// TIA Portal project "CERRADURA" (V11)

(* hardware
DEVICE "S7300/ET200 station_1"  SIMATIC 300-Station
   slot 0: "Perfil soporte_0"  Rail  6ES7 390-1***0-0AA0
   slot 1: "PS 307 2A_1"  PS 307 2A  6ES7 307-1BA00-0AA0
   slot 2: "PLC_1"  CPU 313C-2 DP  6ES7 313-6CF03-0AB0  V2.6
      slot 0: "Interfaz MPI_1"  MPI
      slot 1: "Interfaz DP_1"  DP
      slot 2: "DI16/DO16_1"  DI16/DO16
      slot 4: "Contaje_1"  Counter
   slot 4: "AI4/AO2 x 8bits_1"  AI4/AO2x8/8Bit  6ES7 334-0CE01-0AA0
   slot 5: "CP 343-1 Lean_1"  CP 343-1 LEAN  6GK7 343-1CX10-0XE0  V2.4
   slot 6: "CP 340 RS232C_1"  CP 340 RS232C  6ES7 340-1AH02-0AE0  V1.0
   slot 7: "CP 340 RS422/485_1"  CP 340 RS422/485  6ES7 340-1CH02-0AE0  V1.0
*)

// ===== PLC "PLC_1"  CPU 313C-2 DP =====

VAR_GLOBAL   // PLC tag table "Tabla de variables estándar"
   "1" AT %E0.0 : Bool;
   "2" AT %E0.1 : Bool;
   "3" AT %E0.2 : Bool;
   "4" AT %E0.3 : Bool;
   "5" AT %E0.4 : Bool;
   "6" AT %E0.5 : Bool;
   "7" AT %E0.6 : Bool;
   "8" AT %E0.7 : Bool;
   "9" AT %E1.0 : Bool;
   "0" AT %E1.1 : Bool;
   "#" AT %E1.2 : Bool;
   "*" AT %E1.3 : Bool;
   "Tag_1" AT %AB0 : Byte;
   "Tag_2" AT %AB1 : Byte;
   "Tag_3" AT %AB2 : Byte;
   "Tag_4" AT %AB3 : Byte;
   "Tag_5" AT %M0.0 : Bool;
   "Tag_6" AT %T0 : Timer;
   "Tag_7" AT %A0.0 : Bool;
   "Tag_8" AT %M100.1 : Bool;
   "Tag_9" AT %M100.5 : Bool;
   "Tag_10" AT %A0.1 : Bool;
   "Tag_11" AT %A0.3 : Bool;
   "Tag_12" AT %A3.1 : Bool;
END_VAR

DATA_BLOCK "AUXILIARES"   // DB1
{ S7_Optimized_Access := 'FALSE' }
VERSION : 0.1
   VAR
      FLANCOS : Array [0..70] of Bool;
      BOBINAS : Array [0..70] of Bool;
      REPRESENTACION : Array [0..3] of Byte;
      "CONTADOR H-ACTUAL" : Array [0..2] of Int;
   END_VAR
BEGIN
END_DATA_BLOCK

FUNCTION "DISPLAY UNID. MILLAR." : Void   // FC1, LAD
TITLE = DISPLAY UNIDADES DE MILLAR.
{ S7_Optimized_Access := 'FALSE' }
VERSION : 0.1
// REPRESENTARA EL NUMERO O LETRA CORRESPONDIENTE.
   VAR_OUTPUT
      "UNID. MILLAR" : Byte;
   END_VAR
   VAR_TEMP   // added for the SCL form of the ladder/FBD networks
      _w1 : Bool;
   END_VAR
BEGIN

REGION Network 1: PUESTA EN MARCHA-LETRA "C" HEX. "39"
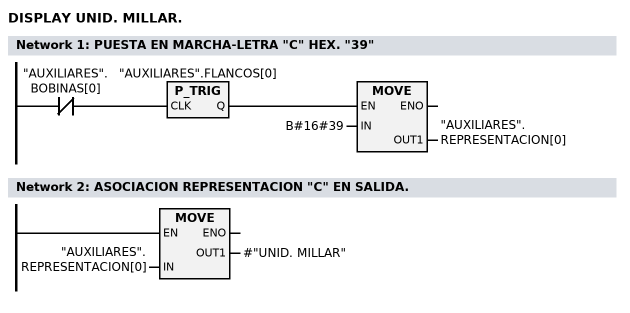
   RUNG wire#powerrail
      I_Contact( "AUXILIARES".BOBINAS[0] )
      P_Trig( "AUXILIARES".FLANCOS[0] )
      { S7_GenerateENO := "TRUE" } Move(in := B#16#39, out1 => "AUXILIARES".REPRESENTACION[0])
   END_RUNG
   // the same network as SCL:
   #_w1 := NOT "AUXILIARES".BOBINAS[0] AND NOT "AUXILIARES".FLANCOS[0];   // rising edge
   "AUXILIARES".FLANCOS[0] := NOT "AUXILIARES".BOBINAS[0];
   IF #_w1 THEN "AUXILIARES".REPRESENTACION[0] := B#16#39; END_IF;
END_REGION

REGION Network 2: ASOCIACION REPRESENTACION "C" EN SALIDA.
   RUNG wire#powerrail
      { S7_GenerateENO := "TRUE" } Move(in := "AUXILIARES".REPRESENTACION[0], out1 => #"UNID. MILLAR")
   END_RUNG
   // the same network as SCL:
   #"UNID. MILLAR" := "AUXILIARES".REPRESENTACION[0];
END_REGION

REGION Network 3: ESTARA REPRESENTADA DURANTE 30 S.
END_REGION

REGION Network 4: CAMBIO DIGITO.
END_REGION
END_FUNCTION

FUNCTION "DISPLAY CENTANAS." : Void   // FC2, LAD
TITLE = DISPLAY CENTANAS.
{ S7_Optimized_Access := 'FALSE' }
VERSION : 0.1
// REPRESENTA EL NUMERO O LETRA CORRESPONDIENTE.
   VAR_OUTPUT
      CENTANAS : Byte;
   END_VAR
   VAR_TEMP   // added for the SCL form of the ladder/FBD networks
      _w1 : Bool;
   END_VAR
BEGIN

REGION Network 1: PUESTA EN MARCHA- "0" HEX. "3F"
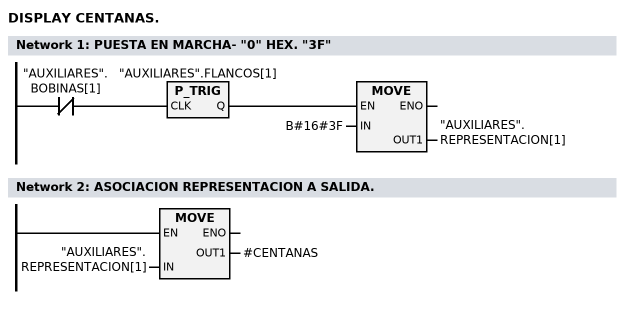
   RUNG wire#powerrail
      I_Contact( "AUXILIARES".BOBINAS[1] )
      P_Trig( "AUXILIARES".FLANCOS[1] )
      { S7_GenerateENO := "TRUE" } Move(in := B#16#3F, out1 => "AUXILIARES".REPRESENTACION[1])
   END_RUNG
   // the same network as SCL:
   #_w1 := NOT "AUXILIARES".BOBINAS[1] AND NOT "AUXILIARES".FLANCOS[1];   // rising edge
   "AUXILIARES".FLANCOS[1] := NOT "AUXILIARES".BOBINAS[1];
   IF #_w1 THEN "AUXILIARES".REPRESENTACION[1] := B#16#3F; END_IF;
END_REGION

REGION Network 2: ASOCIACION REPRESENTACION A SALIDA.
   RUNG wire#powerrail
      { S7_GenerateENO := "TRUE" } Move(in := "AUXILIARES".REPRESENTACION[1], out1 => #CENTANAS)
   END_RUNG
   // the same network as SCL:
   #CENTANAS := "AUXILIARES".REPRESENTACION[1];
END_REGION
END_FUNCTION

FUNCTION "DISPLAY DECENAS" : Void   // FC3, LAD
TITLE = DISPLAY DECENAS.
{ S7_Optimized_Access := 'FALSE' }
VERSION : 0.1
// REPRESENTA EL NUMERO O LETRA CORRESPONDIENTE.
   VAR_OUTPUT
      DECENAS : Byte;
   END_VAR
   VAR_TEMP   // added for the SCL form of the ladder/FBD networks
      _w1 : Bool;
   END_VAR
BEGIN

REGION Network 1: PUESTA EN MARCHA-"D" HEX."5E"
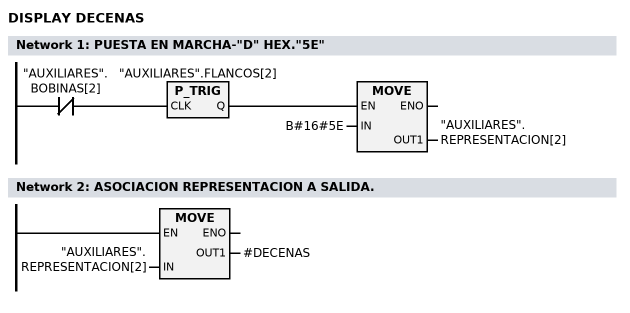
   RUNG wire#powerrail
      I_Contact( "AUXILIARES".BOBINAS[2] )
      P_Trig( "AUXILIARES".FLANCOS[2] )
      { S7_GenerateENO := "TRUE" } Move(in := B#16#5E, out1 => "AUXILIARES".REPRESENTACION[2])
   END_RUNG
   // the same network as SCL:
   #_w1 := NOT "AUXILIARES".BOBINAS[2] AND NOT "AUXILIARES".FLANCOS[2];   // rising edge
   "AUXILIARES".FLANCOS[2] := NOT "AUXILIARES".BOBINAS[2];
   IF #_w1 THEN "AUXILIARES".REPRESENTACION[2] := B#16#5E; END_IF;
END_REGION

REGION Network 2: ASOCIACION REPRESENTACION A SALIDA.
   RUNG wire#powerrail
      { S7_GenerateENO := "TRUE" } Move(in := "AUXILIARES".REPRESENTACION[2], out1 => #DECENAS)
   END_RUNG
   // the same network as SCL:
   #DECENAS := "AUXILIARES".REPRESENTACION[2];
END_REGION
END_FUNCTION

FUNCTION "DISPLAY UNIDADES." : Void   // FC4, LAD
TITLE = DISPLAY UNIDADES
{ S7_Optimized_Access := 'FALSE' }
VERSION : 0.1
// REPRESENTA EL NUMERO O LETRA CORRESPONDIENTE.
   VAR_OUTPUT
      "UNIDADES." : Byte;
   END_VAR
   VAR_TEMP   // added for the SCL form of the ladder/FBD networks
      _w1 : Bool;
   END_VAR
BEGIN

REGION Network 1: PUESTA EN MARCHA-"1" HEX. "6"
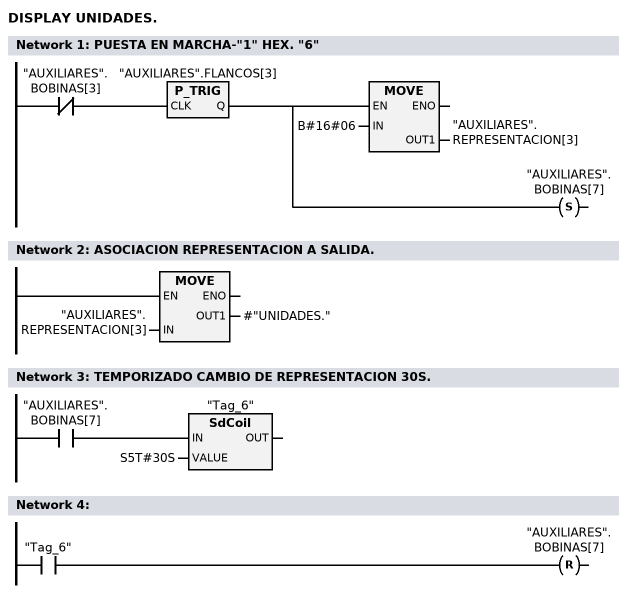
   RUNG wire#powerrail
      I_Contact( "AUXILIARES".BOBINAS[3] )
      P_Trig( "AUXILIARES".FLANCOS[3] )
      wire#w1
      { S7_GenerateENO := "TRUE" } Move(in := B#16#06, out1 => "AUXILIARES".REPRESENTACION[3])
   END_RUNG
   RUNG wire#w1
      S_Coil( "AUXILIARES".BOBINAS[7] )
   END_RUNG
   // the same network as SCL:
   #_w1 := NOT "AUXILIARES".BOBINAS[3] AND NOT "AUXILIARES".FLANCOS[3];   // rising edge
   "AUXILIARES".FLANCOS[3] := NOT "AUXILIARES".BOBINAS[3];
   IF #_w1 THEN
       "AUXILIARES".REPRESENTACION[3] := B#16#06;
       "AUXILIARES".BOBINAS[7] := TRUE;
   END_IF;
END_REGION

REGION Network 2: ASOCIACION REPRESENTACION A SALIDA.
   RUNG wire#powerrail
      { S7_GenerateENO := "TRUE" } Move(in := "AUXILIARES".REPRESENTACION[3], out1 => #"UNIDADES.")
   END_RUNG
   // the same network as SCL:
   #"UNIDADES." := "AUXILIARES".REPRESENTACION[3];
END_REGION

REGION Network 3: TEMPORIZADO CAMBIO DE REPRESENTACION 30S.
   // no SCL statement known for SdCoil: written as a call
   SdCoil(in := "AUXILIARES".BOBINAS[7], value := S5T#30S, operand := "Tag_6");
END_REGION

REGION Network 4
   RUNG wire#powerrail
      Contact( "Tag_6" )
      R_Coil( "AUXILIARES".BOBINAS[7] )
   END_RUNG
   // the same network as SCL:
   IF "Tag_6" THEN "AUXILIARES".BOBINAS[7] := FALSE; END_IF;
END_REGION
END_FUNCTION

FUNCTION "HORA ACTUAL" : Void   // FC5, LAD
TITLE = HORA ACTUAL.
{ S7_Optimized_Access := 'FALSE' }
VERSION : 0.1
// APARECE EN LOS DISPLAY POR ORDEN DE IZQUIERDA A DERECHA EN FORMATO 24 HORAS.SE REPRESENTA DESPUES DE "COD1" Y PERMANECE 60S
   VAR_TEMP   // added for the SCL form of the ladder/FBD networks
      _w1 : Bool;
      _w2 : Bool;
   END_VAR
BEGIN

REGION Network 1: CONTADOR DE SEGUNDOS.
   // MARCA DE CICLO M100.5 1S A 0N -1S A OFF.
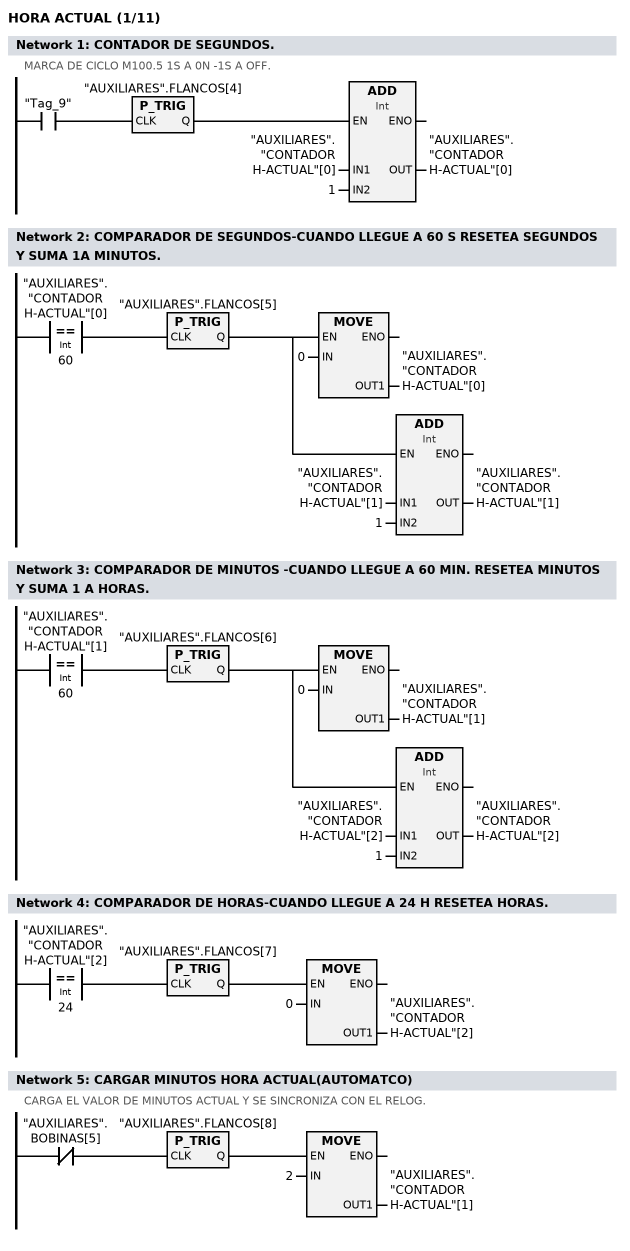
   RUNG wire#powerrail
      Contact( "Tag_9" )
      P_Trig( "AUXILIARES".FLANCOS[4] )
      { S7_Templates := "SrcType := Int"; S7_GenerateENO := "TRUE" } Add(in1 := "AUXILIARES"."CONTADOR H-ACTUAL"[0], in2 := 1, out => "AUXILIARES"."CONTADOR H-ACTUAL"[0])
   END_RUNG
   // the same network as SCL:
   #_w1 := "Tag_9" AND NOT "AUXILIARES".FLANCOS[4];   // rising edge
   "AUXILIARES".FLANCOS[4] := "Tag_9";
   IF #_w1 THEN "AUXILIARES"."CONTADOR H-ACTUAL"[0] := "AUXILIARES"."CONTADOR H-ACTUAL"[0] + 1; END_IF;
END_REGION

REGION Network 2: COMPARADOR DE SEGUNDOS-CUANDO LLEGUE A 60 S RESETEA SEGUNDOS Y SUMA 1A MINUTOS.
   RUNG wire#powerrail
      { S7_Templates := "SrcType := Int" } EQ_Contact(in1 := "AUXILIARES"."CONTADOR H-ACTUAL"[0], in2 := 60)
      P_Trig( "AUXILIARES".FLANCOS[5] )
      wire#w1
      { S7_GenerateENO := "TRUE" } Move(in := 0, out1 => "AUXILIARES"."CONTADOR H-ACTUAL"[0])
   END_RUNG
   RUNG wire#w1
      { S7_Templates := "SrcType := Int"; S7_GenerateENO := "TRUE" } Add(in1 := "AUXILIARES"."CONTADOR H-ACTUAL"[1], in2 := 1, out => "AUXILIARES"."CONTADOR H-ACTUAL"[1])
   END_RUNG
   // the same network as SCL:
   #_w1 := "AUXILIARES"."CONTADOR H-ACTUAL"[0] = 60;
   #_w2 := #_w1 AND NOT "AUXILIARES".FLANCOS[5];   // rising edge
   "AUXILIARES".FLANCOS[5] := #_w1;
   IF #_w2 THEN
       "AUXILIARES"."CONTADOR H-ACTUAL"[0] := 0;
       "AUXILIARES"."CONTADOR H-ACTUAL"[1] := "AUXILIARES"."CONTADOR H-ACTUAL"[1] + 1;
   END_IF;
END_REGION

REGION Network 3: COMPARADOR DE MINUTOS -CUANDO LLEGUE A 60 MIN. RESETEA MINUTOS Y SUMA 1 A HORAS.
   RUNG wire#powerrail
      { S7_Templates := "SrcType := Int" } EQ_Contact(in1 := "AUXILIARES"."CONTADOR H-ACTUAL"[1], in2 := 60)
      P_Trig( "AUXILIARES".FLANCOS[6] )
      wire#w1
      { S7_GenerateENO := "TRUE" } Move(in := 0, out1 => "AUXILIARES"."CONTADOR H-ACTUAL"[1])
   END_RUNG
   RUNG wire#w1
      { S7_Templates := "SrcType := Int"; S7_GenerateENO := "TRUE" } Add(in1 := "AUXILIARES"."CONTADOR H-ACTUAL"[2], in2 := 1, out => "AUXILIARES"."CONTADOR H-ACTUAL"[2])
   END_RUNG
   // the same network as SCL:
   #_w1 := "AUXILIARES"."CONTADOR H-ACTUAL"[1] = 60;
   #_w2 := #_w1 AND NOT "AUXILIARES".FLANCOS[6];   // rising edge
   "AUXILIARES".FLANCOS[6] := #_w1;
   IF #_w2 THEN
       "AUXILIARES"."CONTADOR H-ACTUAL"[1] := 0;
       "AUXILIARES"."CONTADOR H-ACTUAL"[2] := "AUXILIARES"."CONTADOR H-ACTUAL"[2] + 1;
   END_IF;
END_REGION

REGION Network 4: COMPARADOR DE HORAS-CUANDO LLEGUE A 24 H RESETEA HORAS.
   RUNG wire#powerrail
      { S7_Templates := "SrcType := Int" } EQ_Contact(in1 := "AUXILIARES"."CONTADOR H-ACTUAL"[2], in2 := 24)
      P_Trig( "AUXILIARES".FLANCOS[7] )
      { S7_GenerateENO := "TRUE" } Move(in := 0, out1 => "AUXILIARES"."CONTADOR H-ACTUAL"[2])
   END_RUNG
   // the same network as SCL:
   #_w1 := "AUXILIARES"."CONTADOR H-ACTUAL"[2] = 24;
   #_w2 := #_w1 AND NOT "AUXILIARES".FLANCOS[7];   // rising edge
   "AUXILIARES".FLANCOS[7] := #_w1;
   IF #_w2 THEN "AUXILIARES"."CONTADOR H-ACTUAL"[2] := 0; END_IF;
END_REGION

REGION Network 5: CARGAR MINUTOS HORA ACTUAL(AUTOMATCO)
   // CARGA EL VALOR DE MINUTOS ACTUAL Y SE SINCRONIZA CON EL RELOG.
   RUNG wire#powerrail
      I_Contact( "AUXILIARES".BOBINAS[5] )
      P_Trig( "AUXILIARES".FLANCOS[8] )
      { S7_GenerateENO := "TRUE" } Move(in := 2, out1 => "AUXILIARES"."CONTADOR H-ACTUAL"[1])
   END_RUNG
   // the same network as SCL:
   #_w1 := NOT "AUXILIARES".BOBINAS[5] AND NOT "AUXILIARES".FLANCOS[8];   // rising edge
   "AUXILIARES".FLANCOS[8] := NOT "AUXILIARES".BOBINAS[5];
   IF #_w1 THEN "AUXILIARES"."CONTADOR H-ACTUAL"[1] := 2; END_IF;
END_REGION

REGION Network 6: CARGAR HORAS HORA ACTUAL(AUTOMATICO).
   // CARGA EL VALOR DE HORAS ACTUAL Y SE SINCRONIZA CON EL RELOG.
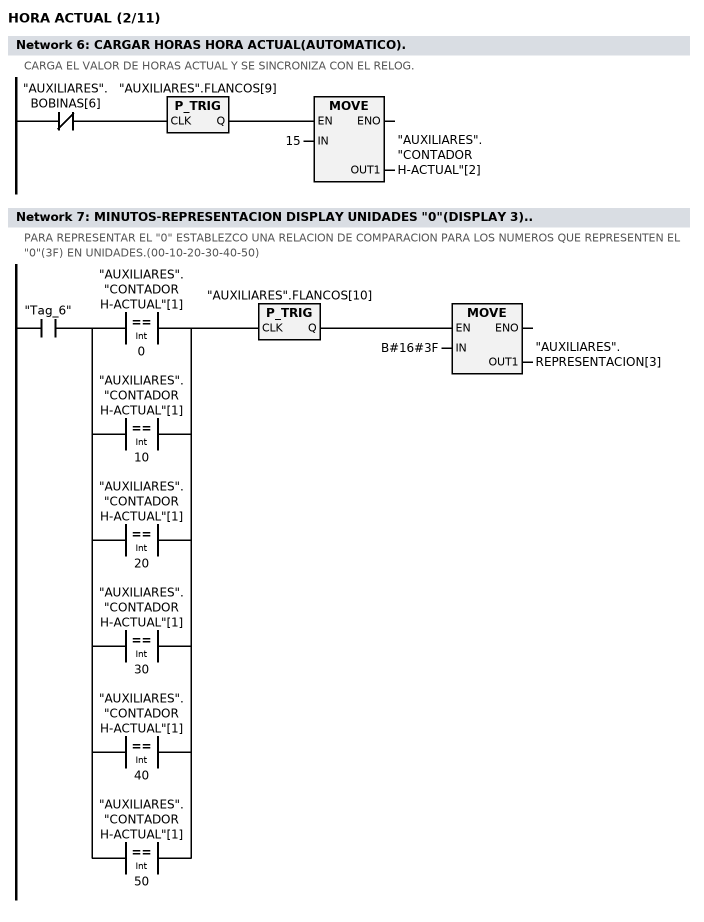
   RUNG wire#powerrail
      I_Contact( "AUXILIARES".BOBINAS[6] )
      P_Trig( "AUXILIARES".FLANCOS[9] )
      { S7_GenerateENO := "TRUE" } Move(in := 15, out1 => "AUXILIARES"."CONTADOR H-ACTUAL"[2])
   END_RUNG
   // the same network as SCL:
   #_w1 := NOT "AUXILIARES".BOBINAS[6] AND NOT "AUXILIARES".FLANCOS[9];   // rising edge
   "AUXILIARES".FLANCOS[9] := NOT "AUXILIARES".BOBINAS[6];
   IF #_w1 THEN "AUXILIARES"."CONTADOR H-ACTUAL"[2] := 15; END_IF;
END_REGION

REGION Network 7: MINUTOS-REPRESENTACION DISPLAY UNIDADES "0"(DISPLAY 3)..
   // PARA REPRESENTAR EL "0" ESTABLEZCO UNA RELACION DE COMPARACION PARA LOS NUMEROS QUE REPRESENTEN EL "0"(3F) EN UNIDADES.(00-10-20-30-40-50)
   RUNG wire#powerrail
      Contact( "Tag_6" )
      wire#w1
      { S7_Templates := "SrcType := Int" } EQ_Contact(in1 := "AUXILIARES"."CONTADOR H-ACTUAL"[1], in2 := 0)
      wire#w2
      P_Trig( "AUXILIARES".FLANCOS[10] )
      { S7_GenerateENO := "TRUE" } Move(in := B#16#3F, out1 => "AUXILIARES".REPRESENTACION[3])
   END_RUNG
   RUNG wire#w1
      { S7_Templates := "SrcType := Int" } EQ_Contact(in1 := "AUXILIARES"."CONTADOR H-ACTUAL"[1], in2 := 10)
   END_RUNG wire#w2
   RUNG wire#w1
      { S7_Templates := "SrcType := Int" } EQ_Contact(in1 := "AUXILIARES"."CONTADOR H-ACTUAL"[1], in2 := 20)
   END_RUNG wire#w2
   RUNG wire#w1
      { S7_Templates := "SrcType := Int" } EQ_Contact(in1 := "AUXILIARES"."CONTADOR H-ACTUAL"[1], in2 := 30)
   END_RUNG wire#w2
   RUNG wire#w1
      { S7_Templates := "SrcType := Int" } EQ_Contact(in1 := "AUXILIARES"."CONTADOR H-ACTUAL"[1], in2 := 40)
   END_RUNG wire#w2
   RUNG wire#w1
      { S7_Templates := "SrcType := Int" } EQ_Contact(in1 := "AUXILIARES"."CONTADOR H-ACTUAL"[1], in2 := 50)
   END_RUNG wire#w2
   // the same network as SCL:
   #_w1 := "Tag_6" AND (("AUXILIARES"."CONTADOR H-ACTUAL"[1] = 0) OR ("AUXILIARES"."CONTADOR H-ACTUAL"[1] = 10) OR ("AUXILIARES"."CONTADOR H-ACTUAL"[1] = 20) OR ("AUXILIARES"."CONTADOR H-ACTUAL"[1] = 30) OR ("AUXILIARES"."CONTADOR H-ACTUAL"[1] = 40) OR ("AUXILIARES"."CONTADOR H-ACTUAL"[1] = 50));
   #_w2 := #_w1 AND NOT "AUXILIARES".FLANCOS[10];   // rising edge
   "AUXILIARES".FLANCOS[10] := #_w1;
   IF #_w2 THEN "AUXILIARES".REPRESENTACION[3] := B#16#3F; END_IF;
END_REGION

REGION Network 8: MINUTOS-REPRESENTACION DISPLAY UNIDADES "1"(DISPLAY 3)..
   // PARA REPRESENTAR EL "1" ESTABLEZCO UNA RELACION DE COMPARACION PARA LOS NUMEROS QUE REPRESENTEN EL "1"(6) EN UNIDADES.(01-11-21-31-41-51)
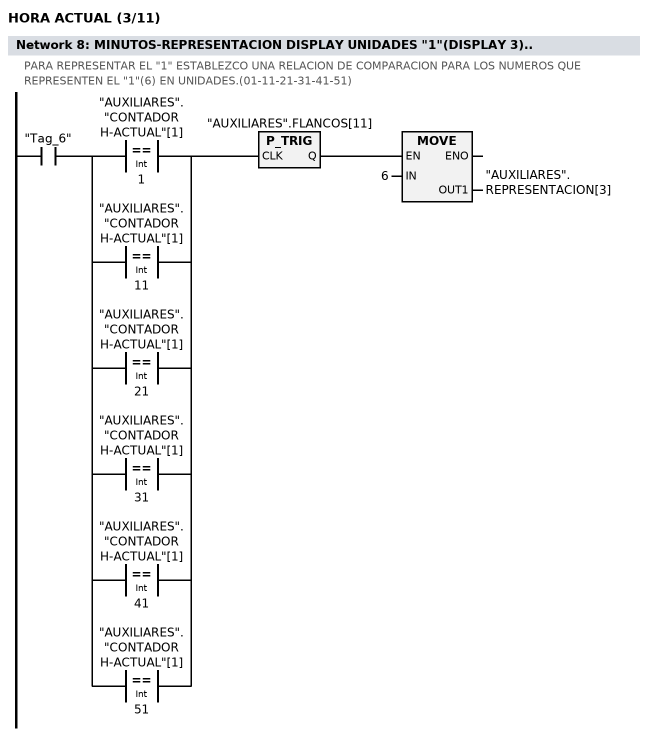
   RUNG wire#powerrail
      Contact( "Tag_6" )
      wire#w1
      { S7_Templates := "SrcType := Int" } EQ_Contact(in1 := "AUXILIARES"."CONTADOR H-ACTUAL"[1], in2 := 1)
      wire#w2
      P_Trig( "AUXILIARES".FLANCOS[11] )
      { S7_GenerateENO := "TRUE" } Move(in := 6, out1 => "AUXILIARES".REPRESENTACION[3])
   END_RUNG
   RUNG wire#w1
      { S7_Templates := "SrcType := Int" } EQ_Contact(in1 := "AUXILIARES"."CONTADOR H-ACTUAL"[1], in2 := 11)
   END_RUNG wire#w2
   RUNG wire#w1
      { S7_Templates := "SrcType := Int" } EQ_Contact(in1 := "AUXILIARES"."CONTADOR H-ACTUAL"[1], in2 := 21)
   END_RUNG wire#w2
   RUNG wire#w1
      { S7_Templates := "SrcType := Int" } EQ_Contact(in1 := "AUXILIARES"."CONTADOR H-ACTUAL"[1], in2 := 31)
   END_RUNG wire#w2
   RUNG wire#w1
      { S7_Templates := "SrcType := Int" } EQ_Contact(in1 := "AUXILIARES"."CONTADOR H-ACTUAL"[1], in2 := 41)
   END_RUNG wire#w2
   RUNG wire#w1
      { S7_Templates := "SrcType := Int" } EQ_Contact(in1 := "AUXILIARES"."CONTADOR H-ACTUAL"[1], in2 := 51)
   END_RUNG wire#w2
   // the same network as SCL:
   #_w1 := "Tag_6" AND (("AUXILIARES"."CONTADOR H-ACTUAL"[1] = 1) OR ("AUXILIARES"."CONTADOR H-ACTUAL"[1] = 11) OR ("AUXILIARES"."CONTADOR H-ACTUAL"[1] = 21) OR ("AUXILIARES"."CONTADOR H-ACTUAL"[1] = 31) OR ("AUXILIARES"."CONTADOR H-ACTUAL"[1] = 41) OR ("AUXILIARES"."CONTADOR H-ACTUAL"[1] = 51));
   #_w2 := #_w1 AND NOT "AUXILIARES".FLANCOS[11];   // rising edge
   "AUXILIARES".FLANCOS[11] := #_w1;
   IF #_w2 THEN "AUXILIARES".REPRESENTACION[3] := 6; END_IF;
END_REGION

REGION Network 9: MINUTOS-REPRESENTACION DISPLAY UNIDADES "2"(DISPLAY 3)..
   // PARA REPRESENTAR EL "2" ESTABLEZCO UNA RELACION DE COMPARACION PARA LOS NUMEROS QUE REPRESENTEN EL "2"(5B) EN UNIDADES.(02-12-22-32-42-52)
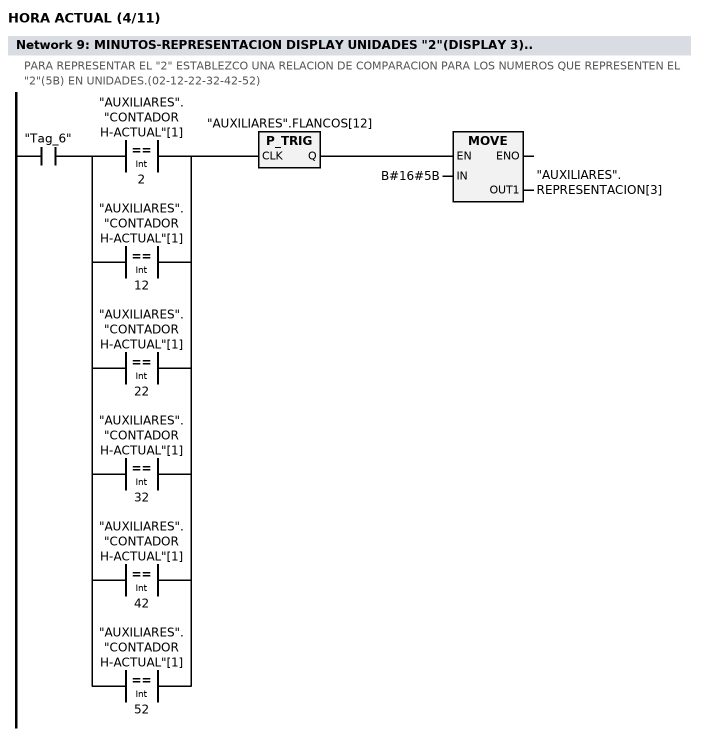
   RUNG wire#powerrail
      Contact( "Tag_6" )
      wire#w1
      { S7_Templates := "SrcType := Int" } EQ_Contact(in1 := "AUXILIARES"."CONTADOR H-ACTUAL"[1], in2 := 2)
      wire#w2
      P_Trig( "AUXILIARES".FLANCOS[12] )
      { S7_GenerateENO := "TRUE" } Move(in := B#16#5B, out1 => "AUXILIARES".REPRESENTACION[3])
   END_RUNG
   RUNG wire#w1
      { S7_Templates := "SrcType := Int" } EQ_Contact(in1 := "AUXILIARES"."CONTADOR H-ACTUAL"[1], in2 := 12)
   END_RUNG wire#w2
   RUNG wire#w1
      { S7_Templates := "SrcType := Int" } EQ_Contact(in1 := "AUXILIARES"."CONTADOR H-ACTUAL"[1], in2 := 22)
   END_RUNG wire#w2
   RUNG wire#w1
      { S7_Templates := "SrcType := Int" } EQ_Contact(in1 := "AUXILIARES"."CONTADOR H-ACTUAL"[1], in2 := 32)
   END_RUNG wire#w2
   RUNG wire#w1
      { S7_Templates := "SrcType := Int" } EQ_Contact(in1 := "AUXILIARES"."CONTADOR H-ACTUAL"[1], in2 := 42)
   END_RUNG wire#w2
   RUNG wire#w1
      { S7_Templates := "SrcType := Int" } EQ_Contact(in1 := "AUXILIARES"."CONTADOR H-ACTUAL"[1], in2 := 52)
   END_RUNG wire#w2
   // the same network as SCL:
   #_w1 := "Tag_6" AND (("AUXILIARES"."CONTADOR H-ACTUAL"[1] = 2) OR ("AUXILIARES"."CONTADOR H-ACTUAL"[1] = 12) OR ("AUXILIARES"."CONTADOR H-ACTUAL"[1] = 22) OR ("AUXILIARES"."CONTADOR H-ACTUAL"[1] = 32) OR ("AUXILIARES"."CONTADOR H-ACTUAL"[1] = 42) OR ("AUXILIARES"."CONTADOR H-ACTUAL"[1] = 52));
   #_w2 := #_w1 AND NOT "AUXILIARES".FLANCOS[12];   // rising edge
   "AUXILIARES".FLANCOS[12] := #_w1;
   IF #_w2 THEN "AUXILIARES".REPRESENTACION[3] := B#16#5B; END_IF;
END_REGION

REGION Network 10: MINUTOS-REPRESENTACION DISPLAY UNIDADES "3"(DISPLAY 3)..
   // PARA REPRESENTAR EL "3" ESTABLEZCO UNA RELACION DE COMPARACION PARA LOS NUMEROS QUE REPRESENTEN EL "3"(4F) EN UNIDADES.(03-13-23-33-43-53)
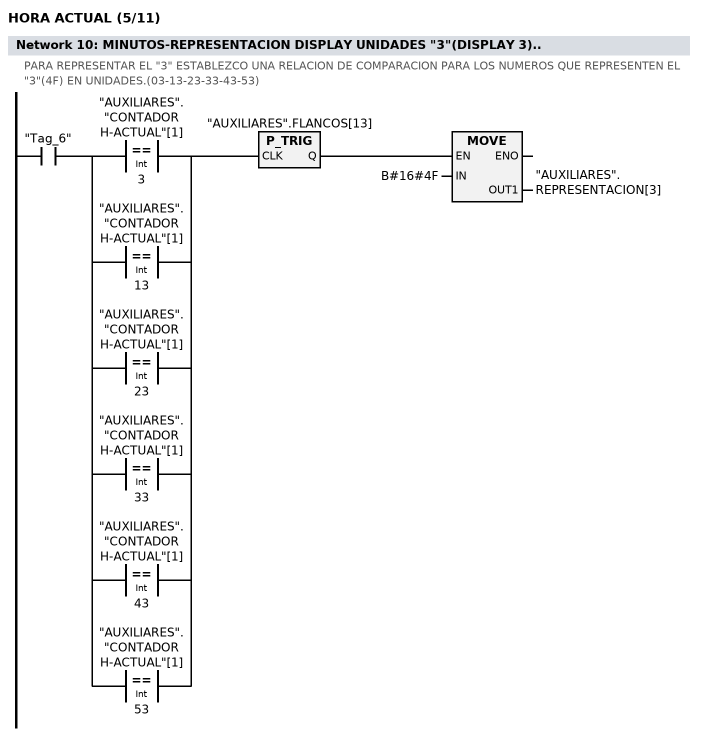
   RUNG wire#powerrail
      Contact( "Tag_6" )
      wire#w1
      { S7_Templates := "SrcType := Int" } EQ_Contact(in1 := "AUXILIARES"."CONTADOR H-ACTUAL"[1], in2 := 3)
      wire#w2
      P_Trig( "AUXILIARES".FLANCOS[13] )
      { S7_GenerateENO := "TRUE" } Move(in := B#16#4F, out1 => "AUXILIARES".REPRESENTACION[3])
   END_RUNG
   RUNG wire#w1
      { S7_Templates := "SrcType := Int" } EQ_Contact(in1 := "AUXILIARES"."CONTADOR H-ACTUAL"[1], in2 := 13)
   END_RUNG wire#w2
   RUNG wire#w1
      { S7_Templates := "SrcType := Int" } EQ_Contact(in1 := "AUXILIARES"."CONTADOR H-ACTUAL"[1], in2 := 23)
   END_RUNG wire#w2
   RUNG wire#w1
      { S7_Templates := "SrcType := Int" } EQ_Contact(in1 := "AUXILIARES"."CONTADOR H-ACTUAL"[1], in2 := 33)
   END_RUNG wire#w2
   RUNG wire#w1
      { S7_Templates := "SrcType := Int" } EQ_Contact(in1 := "AUXILIARES"."CONTADOR H-ACTUAL"[1], in2 := 43)
   END_RUNG wire#w2
   RUNG wire#w1
      { S7_Templates := "SrcType := Int" } EQ_Contact(in1 := "AUXILIARES"."CONTADOR H-ACTUAL"[1], in2 := 53)
   END_RUNG wire#w2
   // the same network as SCL:
   #_w1 := "Tag_6" AND (("AUXILIARES"."CONTADOR H-ACTUAL"[1] = 3) OR ("AUXILIARES"."CONTADOR H-ACTUAL"[1] = 13) OR ("AUXILIARES"."CONTADOR H-ACTUAL"[1] = 23) OR ("AUXILIARES"."CONTADOR H-ACTUAL"[1] = 33) OR ("AUXILIARES"."CONTADOR H-ACTUAL"[1] = 43) OR ("AUXILIARES"."CONTADOR H-ACTUAL"[1] = 53));
   #_w2 := #_w1 AND NOT "AUXILIARES".FLANCOS[13];   // rising edge
   "AUXILIARES".FLANCOS[13] := #_w1;
   IF #_w2 THEN "AUXILIARES".REPRESENTACION[3] := B#16#4F; END_IF;
END_REGION

REGION Network 11: MINUTOS-REPRESENTACION DISPLAY UNIDADES "4"(DISPLAY 3)..
   // PARA REPRESENTAR EL "4" ESTABLEZCO UNA RELACION DE COMPARACION PARA LOS NUMEROS QUE REPRESENTEN EL "4"(66) EN UNIDADES.(04-14-24-34-44-54)
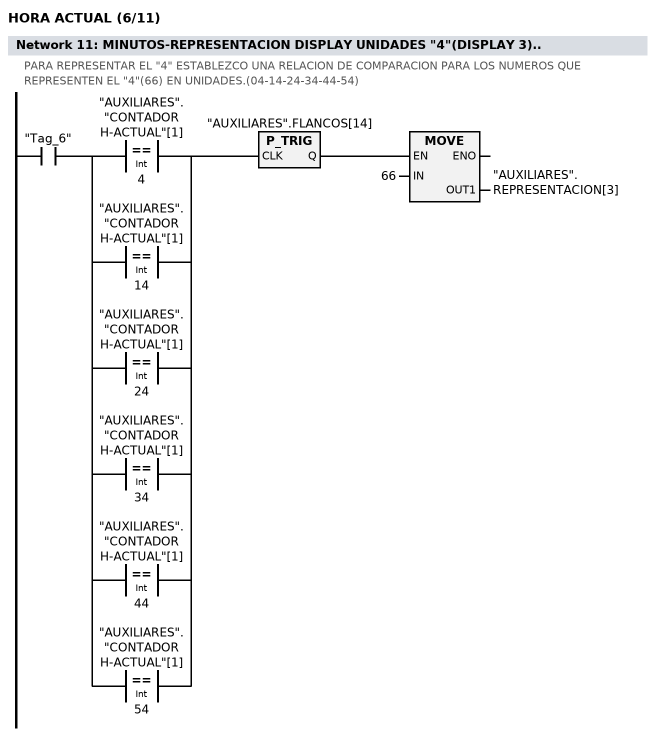
   RUNG wire#powerrail
      Contact( "Tag_6" )
      wire#w1
      { S7_Templates := "SrcType := Int" } EQ_Contact(in1 := "AUXILIARES"."CONTADOR H-ACTUAL"[1], in2 := 4)
      wire#w2
      P_Trig( "AUXILIARES".FLANCOS[14] )
      { S7_GenerateENO := "TRUE" } Move(in := 66, out1 => "AUXILIARES".REPRESENTACION[3])
   END_RUNG
   RUNG wire#w1
      { S7_Templates := "SrcType := Int" } EQ_Contact(in1 := "AUXILIARES"."CONTADOR H-ACTUAL"[1], in2 := 14)
   END_RUNG wire#w2
   RUNG wire#w1
      { S7_Templates := "SrcType := Int" } EQ_Contact(in1 := "AUXILIARES"."CONTADOR H-ACTUAL"[1], in2 := 24)
   END_RUNG wire#w2
   RUNG wire#w1
      { S7_Templates := "SrcType := Int" } EQ_Contact(in1 := "AUXILIARES"."CONTADOR H-ACTUAL"[1], in2 := 34)
   END_RUNG wire#w2
   RUNG wire#w1
      { S7_Templates := "SrcType := Int" } EQ_Contact(in1 := "AUXILIARES"."CONTADOR H-ACTUAL"[1], in2 := 44)
   END_RUNG wire#w2
   RUNG wire#w1
      { S7_Templates := "SrcType := Int" } EQ_Contact(in1 := "AUXILIARES"."CONTADOR H-ACTUAL"[1], in2 := 54)
   END_RUNG wire#w2
   // the same network as SCL:
   #_w1 := "Tag_6" AND (("AUXILIARES"."CONTADOR H-ACTUAL"[1] = 4) OR ("AUXILIARES"."CONTADOR H-ACTUAL"[1] = 14) OR ("AUXILIARES"."CONTADOR H-ACTUAL"[1] = 24) OR ("AUXILIARES"."CONTADOR H-ACTUAL"[1] = 34) OR ("AUXILIARES"."CONTADOR H-ACTUAL"[1] = 44) OR ("AUXILIARES"."CONTADOR H-ACTUAL"[1] = 54));
   #_w2 := #_w1 AND NOT "AUXILIARES".FLANCOS[14];   // rising edge
   "AUXILIARES".FLANCOS[14] := #_w1;
   IF #_w2 THEN "AUXILIARES".REPRESENTACION[3] := 66; END_IF;
END_REGION

REGION Network 12: MINUTOS-REPRESENTACION DISPLAY UNIDADES "5"(DISPLAY 3)..
   // PARA REPRESENTAR EL "5" ESTABLEZCO UNA RELACION DE COMPARACION PARA LOS NUMEROS QUE REPRESENTEN EL "5"(6D) EN UNIDADES.(05-15-25-35-45-55)
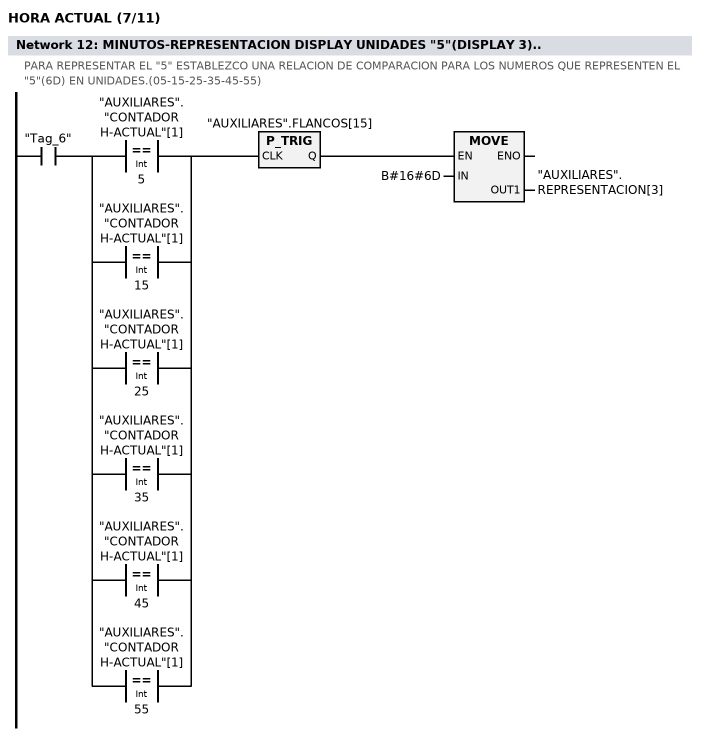
   RUNG wire#powerrail
      Contact( "Tag_6" )
      wire#w1
      { S7_Templates := "SrcType := Int" } EQ_Contact(in1 := "AUXILIARES"."CONTADOR H-ACTUAL"[1], in2 := 5)
      wire#w2
      P_Trig( "AUXILIARES".FLANCOS[15] )
      { S7_GenerateENO := "TRUE" } Move(in := B#16#6D, out1 => "AUXILIARES".REPRESENTACION[3])
   END_RUNG
   RUNG wire#w1
      { S7_Templates := "SrcType := Int" } EQ_Contact(in1 := "AUXILIARES"."CONTADOR H-ACTUAL"[1], in2 := 15)
   END_RUNG wire#w2
   RUNG wire#w1
      { S7_Templates := "SrcType := Int" } EQ_Contact(in1 := "AUXILIARES"."CONTADOR H-ACTUAL"[1], in2 := 25)
   END_RUNG wire#w2
   RUNG wire#w1
      { S7_Templates := "SrcType := Int" } EQ_Contact(in1 := "AUXILIARES"."CONTADOR H-ACTUAL"[1], in2 := 35)
   END_RUNG wire#w2
   RUNG wire#w1
      { S7_Templates := "SrcType := Int" } EQ_Contact(in1 := "AUXILIARES"."CONTADOR H-ACTUAL"[1], in2 := 45)
   END_RUNG wire#w2
   RUNG wire#w1
      { S7_Templates := "SrcType := Int" } EQ_Contact(in1 := "AUXILIARES"."CONTADOR H-ACTUAL"[1], in2 := 55)
   END_RUNG wire#w2
   // the same network as SCL:
   #_w1 := "Tag_6" AND (("AUXILIARES"."CONTADOR H-ACTUAL"[1] = 5) OR ("AUXILIARES"."CONTADOR H-ACTUAL"[1] = 15) OR ("AUXILIARES"."CONTADOR H-ACTUAL"[1] = 25) OR ("AUXILIARES"."CONTADOR H-ACTUAL"[1] = 35) OR ("AUXILIARES"."CONTADOR H-ACTUAL"[1] = 45) OR ("AUXILIARES"."CONTADOR H-ACTUAL"[1] = 55));
   #_w2 := #_w1 AND NOT "AUXILIARES".FLANCOS[15];   // rising edge
   "AUXILIARES".FLANCOS[15] := #_w1;
   IF #_w2 THEN "AUXILIARES".REPRESENTACION[3] := B#16#6D; END_IF;
END_REGION

REGION Network 13: MINUTOS-REPRESENTACION DISPLAY UNIDADES "6"(DISPLAY 3)..
   // PARA REPRESENTAR EL "6" ESTABLEZCO UNA RELACION DE COMPARACION PARA LOS NUMEROS QUE REPRESENTEN EL "6"(7D) EN UNIDADES.(06-16-26-36-46-56)
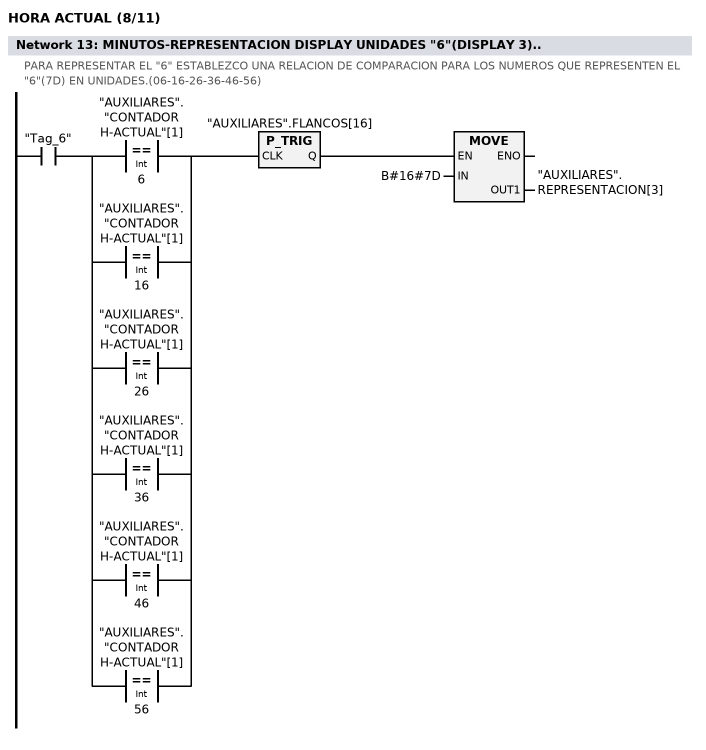
   RUNG wire#powerrail
      Contact( "Tag_6" )
      wire#w1
      { S7_Templates := "SrcType := Int" } EQ_Contact(in1 := "AUXILIARES"."CONTADOR H-ACTUAL"[1], in2 := 6)
      wire#w2
      P_Trig( "AUXILIARES".FLANCOS[16] )
      { S7_GenerateENO := "TRUE" } Move(in := B#16#7D, out1 => "AUXILIARES".REPRESENTACION[3])
   END_RUNG
   RUNG wire#w1
      { S7_Templates := "SrcType := Int" } EQ_Contact(in1 := "AUXILIARES"."CONTADOR H-ACTUAL"[1], in2 := 16)
   END_RUNG wire#w2
   RUNG wire#w1
      { S7_Templates := "SrcType := Int" } EQ_Contact(in1 := "AUXILIARES"."CONTADOR H-ACTUAL"[1], in2 := 26)
   END_RUNG wire#w2
   RUNG wire#w1
      { S7_Templates := "SrcType := Int" } EQ_Contact(in1 := "AUXILIARES"."CONTADOR H-ACTUAL"[1], in2 := 36)
   END_RUNG wire#w2
   RUNG wire#w1
      { S7_Templates := "SrcType := Int" } EQ_Contact(in1 := "AUXILIARES"."CONTADOR H-ACTUAL"[1], in2 := 46)
   END_RUNG wire#w2
   RUNG wire#w1
      { S7_Templates := "SrcType := Int" } EQ_Contact(in1 := "AUXILIARES"."CONTADOR H-ACTUAL"[1], in2 := 56)
   END_RUNG wire#w2
   // the same network as SCL:
   #_w1 := "Tag_6" AND (("AUXILIARES"."CONTADOR H-ACTUAL"[1] = 6) OR ("AUXILIARES"."CONTADOR H-ACTUAL"[1] = 16) OR ("AUXILIARES"."CONTADOR H-ACTUAL"[1] = 26) OR ("AUXILIARES"."CONTADOR H-ACTUAL"[1] = 36) OR ("AUXILIARES"."CONTADOR H-ACTUAL"[1] = 46) OR ("AUXILIARES"."CONTADOR H-ACTUAL"[1] = 56));
   #_w2 := #_w1 AND NOT "AUXILIARES".FLANCOS[16];   // rising edge
   "AUXILIARES".FLANCOS[16] := #_w1;
   IF #_w2 THEN "AUXILIARES".REPRESENTACION[3] := B#16#7D; END_IF;
END_REGION

REGION Network 14: MINUTOS-REPRESENTACION DISPLAY UNIDADES "7"(DISPLAY 3)..
   // PARA REPRESENTAR EL "7" ESTABLEZCO UNA RELACION DE COMPARACION PARA LOS NUMEROS QUE REPRESENTEN EL "7"(7) EN UNIDADES.(07-17-27-37-47-57)
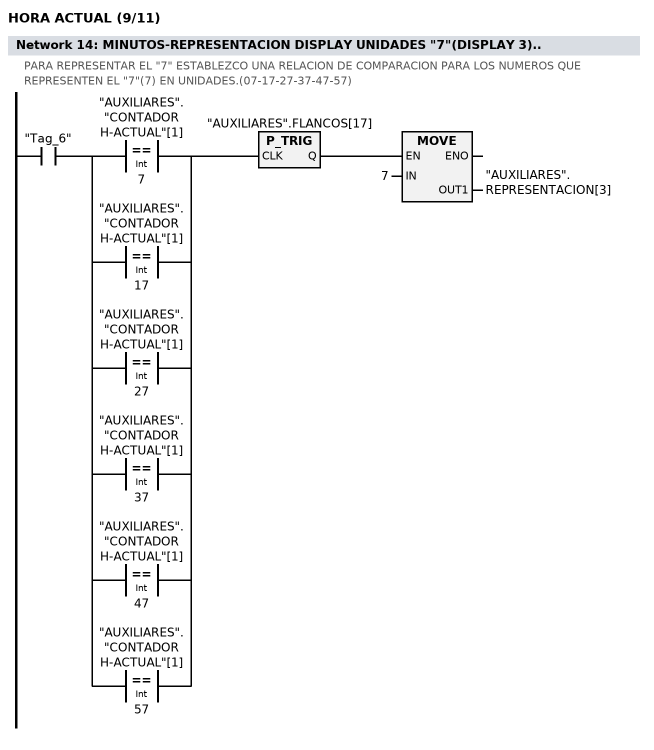
   RUNG wire#powerrail
      Contact( "Tag_6" )
      wire#w1
      { S7_Templates := "SrcType := Int" } EQ_Contact(in1 := "AUXILIARES"."CONTADOR H-ACTUAL"[1], in2 := 7)
      wire#w2
      P_Trig( "AUXILIARES".FLANCOS[17] )
      { S7_GenerateENO := "TRUE" } Move(in := 7, out1 => "AUXILIARES".REPRESENTACION[3])
   END_RUNG
   RUNG wire#w1
      { S7_Templates := "SrcType := Int" } EQ_Contact(in1 := "AUXILIARES"."CONTADOR H-ACTUAL"[1], in2 := 17)
   END_RUNG wire#w2
   RUNG wire#w1
      { S7_Templates := "SrcType := Int" } EQ_Contact(in1 := "AUXILIARES"."CONTADOR H-ACTUAL"[1], in2 := 27)
   END_RUNG wire#w2
   RUNG wire#w1
      { S7_Templates := "SrcType := Int" } EQ_Contact(in1 := "AUXILIARES"."CONTADOR H-ACTUAL"[1], in2 := 37)
   END_RUNG wire#w2
   RUNG wire#w1
      { S7_Templates := "SrcType := Int" } EQ_Contact(in1 := "AUXILIARES"."CONTADOR H-ACTUAL"[1], in2 := 47)
   END_RUNG wire#w2
   RUNG wire#w1
      { S7_Templates := "SrcType := Int" } EQ_Contact(in1 := "AUXILIARES"."CONTADOR H-ACTUAL"[1], in2 := 57)
   END_RUNG wire#w2
   // the same network as SCL:
   #_w1 := "Tag_6" AND (("AUXILIARES"."CONTADOR H-ACTUAL"[1] = 7) OR ("AUXILIARES"."CONTADOR H-ACTUAL"[1] = 17) OR ("AUXILIARES"."CONTADOR H-ACTUAL"[1] = 27) OR ("AUXILIARES"."CONTADOR H-ACTUAL"[1] = 37) OR ("AUXILIARES"."CONTADOR H-ACTUAL"[1] = 47) OR ("AUXILIARES"."CONTADOR H-ACTUAL"[1] = 57));
   #_w2 := #_w1 AND NOT "AUXILIARES".FLANCOS[17];   // rising edge
   "AUXILIARES".FLANCOS[17] := #_w1;
   IF #_w2 THEN "AUXILIARES".REPRESENTACION[3] := 7; END_IF;
END_REGION

REGION Network 15: MINUTOS-REPRESENTACION DISPLAY UNIDADES "8"(DISPLAY 3).....
   // PARA REPRESENTAR EL "8" ESTABLEZCO UNA RELACION DE COMPARACION PARA LOS NUMEROS QUE REPRESENTEN EL "8"(7F) EN UNIDADES.(08-18-28-38-48-58)
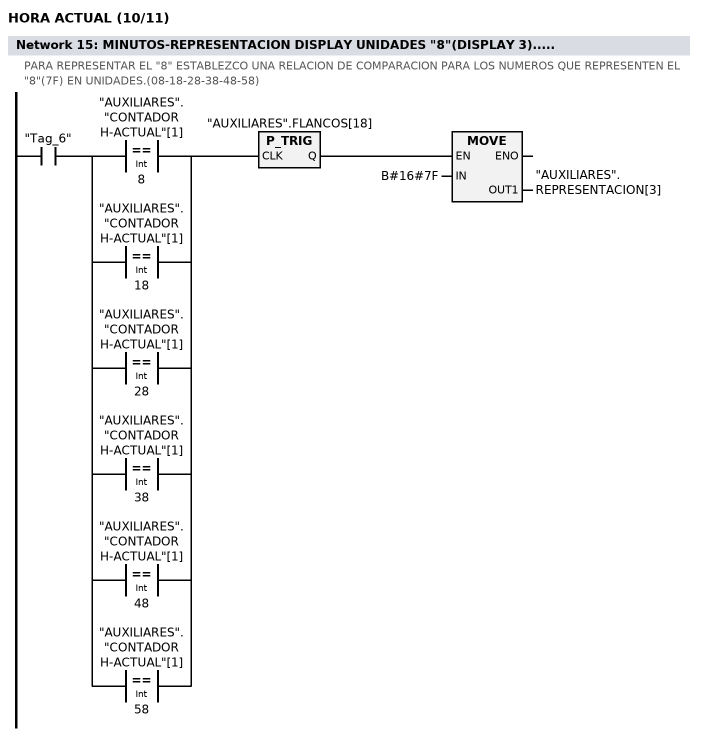
   RUNG wire#powerrail
      Contact( "Tag_6" )
      wire#w1
      { S7_Templates := "SrcType := Int" } EQ_Contact(in1 := "AUXILIARES"."CONTADOR H-ACTUAL"[1], in2 := 8)
      wire#w2
      P_Trig( "AUXILIARES".FLANCOS[18] )
      { S7_GenerateENO := "TRUE" } Move(in := B#16#7F, out1 => "AUXILIARES".REPRESENTACION[3])
   END_RUNG
   RUNG wire#w1
      { S7_Templates := "SrcType := Int" } EQ_Contact(in1 := "AUXILIARES"."CONTADOR H-ACTUAL"[1], in2 := 18)
   END_RUNG wire#w2
   RUNG wire#w1
      { S7_Templates := "SrcType := Int" } EQ_Contact(in1 := "AUXILIARES"."CONTADOR H-ACTUAL"[1], in2 := 28)
   END_RUNG wire#w2
   RUNG wire#w1
      { S7_Templates := "SrcType := Int" } EQ_Contact(in1 := "AUXILIARES"."CONTADOR H-ACTUAL"[1], in2 := 38)
   END_RUNG wire#w2
   RUNG wire#w1
      { S7_Templates := "SrcType := Int" } EQ_Contact(in1 := "AUXILIARES"."CONTADOR H-ACTUAL"[1], in2 := 48)
   END_RUNG wire#w2
   RUNG wire#w1
      { S7_Templates := "SrcType := Int" } EQ_Contact(in1 := "AUXILIARES"."CONTADOR H-ACTUAL"[1], in2 := 58)
   END_RUNG wire#w2
   // the same network as SCL:
   #_w1 := "Tag_6" AND (("AUXILIARES"."CONTADOR H-ACTUAL"[1] = 8) OR ("AUXILIARES"."CONTADOR H-ACTUAL"[1] = 18) OR ("AUXILIARES"."CONTADOR H-ACTUAL"[1] = 28) OR ("AUXILIARES"."CONTADOR H-ACTUAL"[1] = 38) OR ("AUXILIARES"."CONTADOR H-ACTUAL"[1] = 48) OR ("AUXILIARES"."CONTADOR H-ACTUAL"[1] = 58));
   #_w2 := #_w1 AND NOT "AUXILIARES".FLANCOS[18];   // rising edge
   "AUXILIARES".FLANCOS[18] := #_w1;
   IF #_w2 THEN "AUXILIARES".REPRESENTACION[3] := B#16#7F; END_IF;
END_REGION

REGION Network 16: MINUTOS-REPRESENTACION DISPLAY UNIDADES "9"(DISPLAY 3)..
   // PARA REPRESENTAR EL "9" ESTABLEZCO UNA RELACION DE COMPARACION PARA LOS NUMEROS QUE REPRESENTEN EL "9"(6F) EN UNIDADES.(09-19-29-39-49-59)
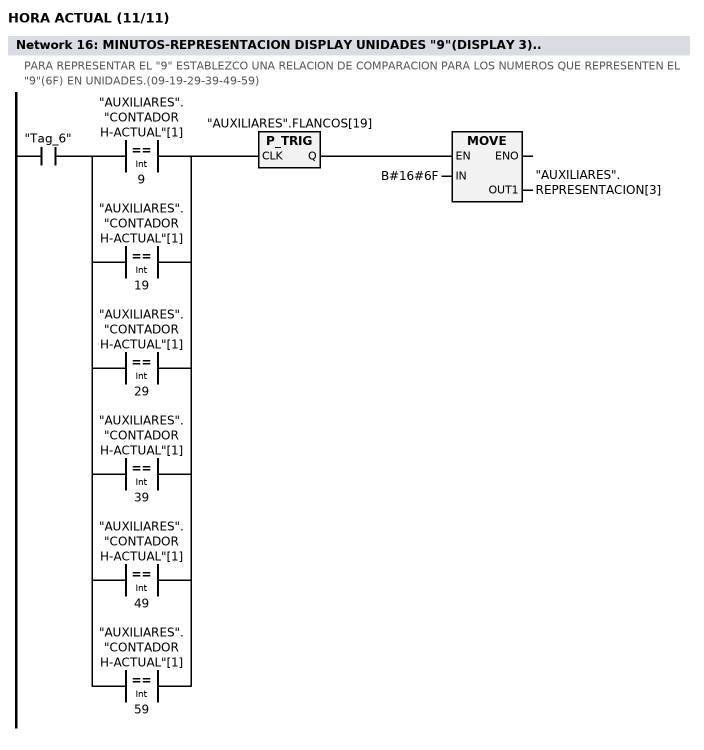
   RUNG wire#powerrail
      Contact( "Tag_6" )
      wire#w1
      { S7_Templates := "SrcType := Int" } EQ_Contact(in1 := "AUXILIARES"."CONTADOR H-ACTUAL"[1], in2 := 9)
      wire#w2
      P_Trig( "AUXILIARES".FLANCOS[19] )
      { S7_GenerateENO := "TRUE" } Move(in := B#16#6F, out1 => "AUXILIARES".REPRESENTACION[3])
   END_RUNG
   RUNG wire#w1
      { S7_Templates := "SrcType := Int" } EQ_Contact(in1 := "AUXILIARES"."CONTADOR H-ACTUAL"[1], in2 := 19)
   END_RUNG wire#w2
   RUNG wire#w1
      { S7_Templates := "SrcType := Int" } EQ_Contact(in1 := "AUXILIARES"."CONTADOR H-ACTUAL"[1], in2 := 29)
   END_RUNG wire#w2
   RUNG wire#w1
      { S7_Templates := "SrcType := Int" } EQ_Contact(in1 := "AUXILIARES"."CONTADOR H-ACTUAL"[1], in2 := 39)
   END_RUNG wire#w2
   RUNG wire#w1
      { S7_Templates := "SrcType := Int" } EQ_Contact(in1 := "AUXILIARES"."CONTADOR H-ACTUAL"[1], in2 := 49)
   END_RUNG wire#w2
   RUNG wire#w1
      { S7_Templates := "SrcType := Int" } EQ_Contact(in1 := "AUXILIARES"."CONTADOR H-ACTUAL"[1], in2 := 59)
   END_RUNG wire#w2
   // the same network as SCL:
   #_w1 := "Tag_6" AND (("AUXILIARES"."CONTADOR H-ACTUAL"[1] = 9) OR ("AUXILIARES"."CONTADOR H-ACTUAL"[1] = 19) OR ("AUXILIARES"."CONTADOR H-ACTUAL"[1] = 29) OR ("AUXILIARES"."CONTADOR H-ACTUAL"[1] = 39) OR ("AUXILIARES"."CONTADOR H-ACTUAL"[1] = 49) OR ("AUXILIARES"."CONTADOR H-ACTUAL"[1] = 59));
   #_w2 := #_w1 AND NOT "AUXILIARES".FLANCOS[19];   // rising edge
   "AUXILIARES".FLANCOS[19] := #_w1;
   IF #_w2 THEN "AUXILIARES".REPRESENTACION[3] := B#16#6F; END_IF;
END_REGION
END_FUNCTION

ORGANIZATION_BLOCK "Main"   // OB1, LAD
TITLE = CERRADURA PROGRAMABLE. / "Main Program Sweep (Cycle)"
{ S7_Optimized_Access := 'FALSE' }
VERSION : 0.1
   VAR_TEMP
      OB1_EV_CLASS : Byte;   // Bits 0-3 = 1 (Coming event), Bits 4-7 = 1 (Event class 1)
      OB1_SCAN_1 : Byte;   // 1 (Cold restart scan 1 of OB 1), 3 (Scan 2-n of OB 1)
      OB1_PRIORITY : Byte;   // Priority of OB Execution
      OB1_OB_NUMBR : Byte;   // 1 (Organization block 1, OB1)
      OB1_RESERVED_1 : Byte;   // Reserved for system
      OB1_RESERVED_2 : Byte;   // Reserved for system
      OB1_PREV_CYCLE : Int;   // Cycle time of previous OB1 scan (milliseconds)
      OB1_MIN_CYCLE : Int;   // Minimum cycle time of OB1 (milliseconds)
      OB1_MAX_CYCLE : Int;   // Maximum cycle time of OB1 (milliseconds)
      OB1_DATE_TIME : Date_And_Time;   // Date and time OB1 started
   END_VAR
BEGIN

REGION Network 1: DIGITO UNIDADES DE MILLAR.
   // REPRESENTARA EL DIGITO QUE PROCEDA.PUESTA EM MARCHA "C".
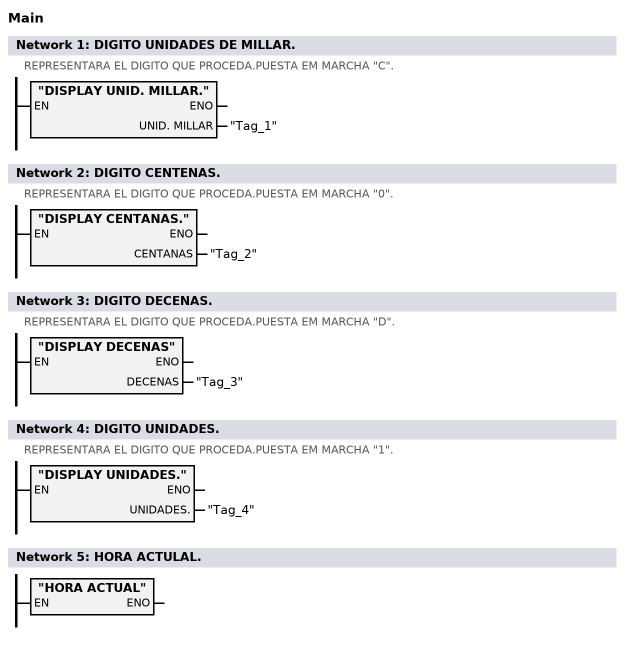
   RUNG wire#powerrail
      "DISPLAY UNID. MILLAR."("UNID. MILLAR" => "Tag_1")
   END_RUNG
   // the same network as SCL:
   "DISPLAY UNID. MILLAR."("UNID. MILLAR" => "Tag_1");
END_REGION

REGION Network 2: DIGITO CENTENAS.
   // REPRESENTARA EL DIGITO QUE PROCEDA.PUESTA EM MARCHA "0".
   RUNG wire#powerrail
      "DISPLAY CENTANAS."(CENTANAS => "Tag_2")
   END_RUNG
   // the same network as SCL:
   "DISPLAY CENTANAS."(CENTANAS => "Tag_2");
END_REGION

REGION Network 3: DIGITO DECENAS.
   // REPRESENTARA EL DIGITO QUE PROCEDA.PUESTA EM MARCHA "D".
   RUNG wire#powerrail
      "DISPLAY DECENAS"(DECENAS => "Tag_3")
   END_RUNG
   // the same network as SCL:
   "DISPLAY DECENAS"(DECENAS => "Tag_3");
END_REGION

REGION Network 4: DIGITO UNIDADES.
   // REPRESENTARA EL DIGITO QUE PROCEDA.PUESTA EM MARCHA "1".
   RUNG wire#powerrail
      "DISPLAY UNIDADES."("UNIDADES." => "Tag_4")
   END_RUNG
   // the same network as SCL:
   "DISPLAY UNIDADES."("UNIDADES." => "Tag_4");
END_REGION

REGION Network 5: HORA ACTULAL.
   RUNG wire#powerrail
      "HORA ACTUAL"()
   END_RUNG
   // the same network as SCL:
   "HORA ACTUAL"();
END_REGION
END_ORGANIZATION_BLOCK